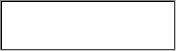
VISUALIZATION VISU_HMI_ROUTINES_BUTTON  // 176x51
VAR_IN_OUT
    m_Hmi : FB_HMI_BUTTON;
END_VAR
    Rectangle (0,0 175x50), invisible if: m_Hmi.bIsNotOrange
    Rectangle (0,0 175x50), invisible if: m_Hmi.bIsNotGray
    Rectangle (0,0 175x50), invisible if: m_Hmi.bIsNotBlue
    Rectangle (0,0 175x50), invisible if: m_Hmi.bIsNotRed
    Rectangle (0,0 175x50), invisible if: m_Hmi.bIsNotGreen
    Rectangle (0,0 175x50), "%s", text variable: m_Hmi.sName
    Rectangle (0,0 175x50), invisible if: m_Hmi.bNotActivated
    Line (0,49) (175,49), invisible if: m_Hmi.bActivated
    Line (174,0) (174,50), invisible if: m_Hmi.bActivated
    Line (174,0) (0,0), invisible if: m_Hmi.bActivated
    Line (0,49) (0,0), invisible if: m_Hmi.bActivated
    Line (175,50) (175,1), invisible if: m_Hmi.bNotActivated
    Line (0,1) (174,1), invisible if: m_Hmi.bNotActivated
    Line (1,0) (1,49), invisible if: m_Hmi.bNotActivated
    Line (175,50) (1,50), invisible if: m_Hmi.bNotActivated
END_VISUALIZATION

(* stored: Version 1.1.0.1, ProductVersion 3.1.4024.14
   Visu VISU_HMI_ROUTINES_BUTTON: Id {d946574d-689f-437e-b8b0-5aa6d270eda9} *)
